// Mitsubishi GX Works2 project: 26   PLC: FX3G

// task Task_01 (event TRUE, interval 0, priority 31): POU_01

PROGRAM POU_01
VAR
  gas : INT;
  ton1 : TON;
  gas2 : BOOL;
  ton2 : TON;
  gas3 : INT;
END_VAR
IF M8002 THEN
	gas := 0;
	gas3:=0;
END_IF;

ton2(IN := gas2, PT := T#20s);
	IF ton2.Q THEN
		gas:=0;
		gas2:=FALSE;
		gas3:=0;
	END_IF;

CASE gas3 OF
	
	1:
	IF M2 THEN
	Y2:=TRUE;
END_IF;

IF M3  THEN
	Y3:=TRUE;
	END_IF;
END_CASE;



CASE gas OF
0:
Y0:=FALSE;
Y1:=FALSE;
Y2:=FALSE;
Y3:=FALSE;
Y4:=FALSE;
Y5:=FALSE;
Y6:=FALSE;
IF M6=TRUE THEN
	gas:=1;
END_IF;


1:
IF M4 THEN
	gas:=11;
	Y6:=TRUE;
END_IF;

IF M5=TRUE THEN
	gas:=21;
	Y5:=TRUE;
END_IF;


11:
IF M0  THEN
	gas2 := TRUE;
   gas3:=1;
END_IF;


IF ton2.Q THEN
	gas2 :=0;
END_IF;
 

21:
IF M0=TRUE THEN
	gas:=22;
END_IF;

22:
Y2:=TRUE;
ton1(IN := NOT ton1.Q, PT := T#5s);
	IF ton1.Q THEN
		Y2:=FALSE;
		gas:=23;
	END_IF;

23:
Y3:=TRUE;
ton1(IN := NOT ton1.Q, PT := T#5s);
	IF ton1.Q THEN
		Y3:=FALSE;
		gas:=24;
	END_IF;
	
24:
Y4:=TRUE;
ton1(IN := NOT ton1.Q, PT := T#10s);
	IF ton1.Q THEN
		gas:=0;
		Y4:=FALSE;
	END_IF;
END_CASE;
;
END_PROGRAM
